(* PLC project Test.project, CODESYS CODESYS V3.5 SP21 Patch 5 *)
(* stored: creationDateTime 2026-05-07T14:55:41.6791703, modificationDateTime 2026-05-07T14:54:46.6861198 *)

PROGRAM PLC_PRG
  VAR
    counter : INT;
  END_VAR

                    
counter := counter + 1;

IF counter > 100 THEN
	counter := 0;
END_IF

                  
END_PROGRAM

CONFIGURATION Device
  RESOURCE Application ON PLC
    VAR_GLOBAL  (* Device *)
      Processor_Load_Lower_Limit : DWORD := 80;
      Processor_Load_Upper_Limit : DWORD := 90;  (* Processor Load Lower Limit *)
      Processor_Load_Processor_Share : DWORD := 90;  (* Processor Load Upper Limit *)
      Processor_Load_Should_Throw_ProcessorLoadWatchdog_Exception : BOOL := FALSE;  (* Processor Load Processor Share *)
      TCM_control : UDINT := 16777216;
      k_bus_cycle_time : WORD := 10;  (* TCM control | 0: disable / TCM version (16777216 = 01.00.00.00) enable *)
      program_start_interlock : BOOL := TRUE;  (* k-bus cycle time | cycle time in [ms] *)
    END_VAR
    TASK MainTask(INTERVAL := T#50ms, PRIORITY := 15);
    PROGRAM PLC_PRG WITH MainTask : PLC_PRG;
  END_RESOURCE
END_CONFIGURATION

CONFIGURATION Kbus
END_CONFIGURATION

CONFIGURATION Serial
END_CONFIGURATION

CONFIGURATION COM1
END_CONFIGURATION
